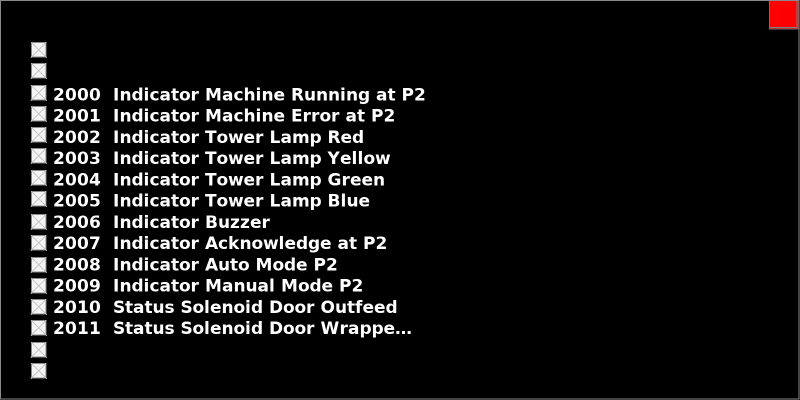
VISUALIZATION P2_DO1  // 800x400, background image 
    ImageSwitcher (31,42 15x15), variable: InputOutput_GVL.Digital_Output[1], behaviour: TOGGLE
    Label (50,16 625x391), "2000 Indicator Machine Running at P2 2001 Indicator Machine Error at P2 2002 Indicator Tower Lamp Red 2003 Indicator Tower Lamp Yellow 2004 Indicator Tower Lamp Green 2005 Indicator Tower Lamp Blue 2006 Indicator Buzzer 2007 Indicator Acknowledge at P2 2008 Indicator Auto Mode P2 2009 Indicator Manual Mode P2 2010 Status Solenoid Door Outfeed 2011 Status Solenoid Door Wrapper 2012 2013 Pneumatic Stopper Modullar Adv 2014 Pneumatic Stopper Modullar Rtc 2015 Move Forward for Loaded Pallet Outfeed Roller Conveyor 5"
    ImageSwitcher (31,63 15x15), variable: InputOutput_GVL.Digital_Output[2], behaviour: TOGGLE
    ImageSwitcher (31,85 15x15), variable: InputOutput_GVL.Digital_Output[3], behaviour: TOGGLE
    ImageSwitcher (31,106 15x15), variable: InputOutput_GVL.Digital_Output[4], behaviour: TOGGLE
    ImageSwitcher (31,127 15x15), variable: InputOutput_GVL.Digital_Output[5], behaviour: TOGGLE
    ImageSwitcher (31,148 15x15), variable: InputOutput_GVL.Digital_Output[6], behaviour: TOGGLE
    ImageSwitcher (31,170 15x15), variable: InputOutput_GVL.Digital_Output[7], behaviour: TOGGLE
    ImageSwitcher (31,191 15x15), variable: InputOutput_GVL.Digital_Output[8], behaviour: TOGGLE
    ImageSwitcher (31,214 15x15), variable: InputOutput_GVL.Digital_Output[9], behaviour: TOGGLE
    ImageSwitcher (31,235 15x15), variable: InputOutput_GVL.Digital_Output[10], behaviour: TOGGLE
    ImageSwitcher (31,257 15x15), variable: InputOutput_GVL.Digital_Output[11], behaviour: TOGGLE
    ImageSwitcher (31,278 15x15), variable: InputOutput_GVL.Digital_Output[12], behaviour: TOGGLE
    ImageSwitcher (31,299 15x15), variable: InputOutput_GVL.Digital_Output[13], behaviour: TOGGLE
    ImageSwitcher (31,320 15x15), variable: InputOutput_GVL.Digital_Output[14], behaviour: TOGGLE
    ImageSwitcher (31,342 15x15), variable: InputOutput_GVL.Digital_Output[15], behaviour: TOGGLE
    ImageSwitcher (31,363 15x15), variable: InputOutput_GVL.Digital_Output[16], behaviour: TOGGLE
    Button (769,-1 30x30), image: VisuSymbols.Symbols.Wrong
        OnMouseClick: CloseDialog Dialog=P2_DO1, Result=OK, NumpadKeypadSet=True
END_VISUALIZATION

(* stored: Version 1.1.0.1, ProductVersion 3.1.4024.12
   Visu P2_DO1: Id {d42b3704-bd8f-4c39-bed5-688956b606f4} *)
